(*******************************************************************************
                          protoc-gen-twincat V0.0.0.0                           
             https://github.bhs-world.com/CorrML/protoc-gen-twincat             
*******************************************************************************)
{attribute 'no_explicit_call' := 'do not call this POU directly'}
{attribute 'no-analysis'}
FUNCTION_BLOCK INTERNAL FINAL FB_ScalarTypes IMPLEMENTS I_Message
VAR
    _fbMessageParser : FB_MessageParser(ipMessage:= THIS^);
    _fbMessageWriter : FB_MessageWriter(ipMessage:= THIS^);
    _stScalarTypes : ST_ScalarTypes;
    END_VAR

{attribute 'no-analysis'}
(* Calculates the size of this message in Protocol Buffer wire format, in bytes. *)
METHOD CalculateSize : UDINT
VAR
    nSize : UDINT;
    nRepeatedFieldSize : UDINT;
END_VAR
// double double_value = 1;
nSize := nSize + 1 + F_ComputeDoubleSize(fValue:= _stScalarTypes.double_value);
// float float_value = 2;
nSize := nSize + 1 + F_ComputeFloatSize(fValue:= _stScalarTypes.float_value);
// int32 int32_value = 3;
nSize := nSize + 1 + F_ComputeInt32Size(anyDint:= _stScalarTypes.int32_value);
// int32 int32_value_as_word = 30;
nSize := nSize + 2 + F_ComputeInt32Size(anyDint:= _stScalarTypes.int32_value_as_word);
// int64 int64_value = 4;
nSize := nSize + 1 + F_ComputeInt64Size(anyLint:= _stScalarTypes.int64_value);
// int64 int64_value_as_dint = 40;
nSize := nSize + 2 + F_ComputeInt64Size(anyLint:= _stScalarTypes.int64_value_as_dint);
// uint32 uint32_value = 5;
nSize := nSize + 1 + F_ComputeUint32Size(anyUdint:= _stScalarTypes.uint32_value);
// uint32 uint32_value_as_byte = 50;
nSize := nSize + 2 + F_ComputeUint32Size(anyUdint:= _stScalarTypes.uint32_value_as_byte);
// uint64 uint64_value = 6;
nSize := nSize + 1 + F_ComputeUint64Size(anyUlint:= _stScalarTypes.uint64_value);
// uint64 uint64_value_as_dword = 60;
nSize := nSize + 2 + F_ComputeUint64Size(anyUlint:= _stScalarTypes.uint64_value_as_dword);
// sint32 sint32_value = 7;
nSize := nSize + 1 + F_ComputeSint32Size(anyDint:= _stScalarTypes.sint32_value);
// sint64 sint64_value = 8;
nSize := nSize + 1 + F_ComputeSint64Size(anyLint:= _stScalarTypes.sint64_value);
// fixed32 fixed32_value = 9;
nSize := nSize + 1 + F_ComputeFixed32Size(nValue:= _stScalarTypes.fixed32_value);
// fixed64 fixed64_value = 10;
nSize := nSize + 1 + F_ComputeFixed64Size(nValue:= _stScalarTypes.fixed64_value);
// sfixed32 sfixed32_value = 11;
nSize := nSize + 1 + F_ComputeSfixed32Size(nValue:= _stScalarTypes.sfixed32_value);
// sfixed64 sfixed64_value = 12;
nSize := nSize + 1 + F_ComputeSfixed64Size(nValue:= _stScalarTypes.sfixed64_value);
// bool bool_value = 13;
nSize := nSize + 1 + F_ComputeBoolSize(bValue:= _stScalarTypes.bool_value);
// string string_value = 14;
nSize := nSize + 1 + F_ComputeStringSize(anyString:= _stScalarTypes.string_value);
// bytes bytes_value = 15;
nSize := nSize + 1 + F_ComputeBytesSize(aBytes:= _stScalarTypes.bytes_value, nCount:= _stScalarTypes.bytes_value_count);
CalculateSize := nSize;
END_METHOD

(* Merges the data from the specified coded input stream with the current message.*)
METHOD MergeFrom : HRESULT
VAR_IN_OUT
    fbParseCtx : FB_ParseContext;
END_VAR
VAR
    nTag : UDINT;
END_VAR
REPEAT
MergeFrom := fbParseCtx.ReadTag(nTag=> nTag);
IF SUCCEEDED(MergeFrom) AND nTag = 0 THEN
    EXIT;
END_IF;

IF FAILED(MergeFrom) THEN
    RETURN;
END_IF

CASE nTag OF
    16#09:    // double double_value = 1;
        MergeFrom := fbParseCtx.ReadDouble(fValue=> _stScalarTypes.double_value); 
    16#15:    // float float_value = 2;
        MergeFrom := fbParseCtx.ReadFloat(fValue=> _stScalarTypes.float_value); 
    16#18:    // int32 int32_value = 3;
        MergeFrom := fbParseCtx.ReadInt32(anyDint:= _stScalarTypes.int32_value); 
    16#F0:    // int32 int32_value_as_word = 30;
        MergeFrom := fbParseCtx.ReadInt32(anyDint:= _stScalarTypes.int32_value_as_word); 
    16#20:    // int64 int64_value = 4;
        MergeFrom := fbParseCtx.ReadInt64(anyLint:= _stScalarTypes.int64_value); 
    16#140:    // int64 int64_value_as_dint = 40;
        MergeFrom := fbParseCtx.ReadInt64(anyLint:= _stScalarTypes.int64_value_as_dint); 
    16#28:    // uint32 uint32_value = 5;
        MergeFrom := fbParseCtx.ReadUint32(anyUdint:= _stScalarTypes.uint32_value); 
    16#190:    // uint32 uint32_value_as_byte = 50;
        MergeFrom := fbParseCtx.ReadUint32(anyUdint:= _stScalarTypes.uint32_value_as_byte); 
    16#30:    // uint64 uint64_value = 6;
        MergeFrom := fbParseCtx.ReadUint64(anyUlint:= _stScalarTypes.uint64_value); 
    16#1E0:    // uint64 uint64_value_as_dword = 60;
        MergeFrom := fbParseCtx.ReadUint64(anyUlint:= _stScalarTypes.uint64_value_as_dword); 
    16#38:    // sint32 sint32_value = 7;
        MergeFrom := fbParseCtx.ReadSint32(anyDint:= _stScalarTypes.sint32_value); 
    16#40:    // sint64 sint64_value = 8;
        MergeFrom := fbParseCtx.ReadSint64(anyLint:= _stScalarTypes.sint64_value); 
    16#4D:    // fixed32 fixed32_value = 9;
        MergeFrom := fbParseCtx.ReadFixed32(nValue=> _stScalarTypes.fixed32_value); 
    16#51:    // fixed64 fixed64_value = 10;
        MergeFrom := fbParseCtx.ReadFixed64(nValue=> _stScalarTypes.fixed64_value); 
    16#5D:    // sfixed32 sfixed32_value = 11;
        MergeFrom := fbParseCtx.ReadSfixed32(nValue=> _stScalarTypes.sfixed32_value); 
    16#61:    // sfixed64 sfixed64_value = 12;
        MergeFrom := fbParseCtx.ReadSfixed64(nValue=> _stScalarTypes.sfixed64_value); 
    16#68:    // bool bool_value = 13;
        MergeFrom := fbParseCtx.ReadBool(bValue=> _stScalarTypes.bool_value); 
    16#72:    // string string_value = 14;
        MergeFrom := fbParseCtx.ReadString(anyStringOut:= _stScalarTypes.string_value); 
    16#7A:    // bytes bytes_value = 15;
        MergeFrom := fbParseCtx.ReadBytes(aBytes:= _stScalarTypes.bytes_value, nCount=> _stScalarTypes.bytes_value_count); 
ELSE
    MergeFrom := fbParseCtx.SkipLastField();
END_CASE

UNTIL (FAILED(MergeFrom) OR nTag = 0)
END_REPEAT
END_METHOD

PROPERTY PUBLIC MessageValue : T_Any
GET
MessageValue := F_ToAnyType(anyArg:= _stScalarTypes);
END_GET
END_PROPERTY

PROPERTY PUBLIC Parser : REFERENCE TO FB_MessageParser
GET
Parser REF= THIS^._fbMessageParser;
END_GET
END_PROPERTY

PROPERTY PUBLIC ScalarTypes : ST_ScalarTypes
GET
ScalarTypes := _stScalarTypes;
END_GET
SET
_stScalarTypes := ScalarTypes;
END_SET
END_PROPERTY

(* Writer for this message.*)
PROPERTY PUBLIC Writer : REFERENCE TO FB_MessageWriter
GET
Writer REF= THIS^._fbMessageWriter;
END_GET
END_PROPERTY

(* Writes the data to the given coded output stream.*)
METHOD WriteTo : HRESULT
VAR_IN_OUT
	(* Coded output stream to write the data to. *)
	fbWriteCtx	: FB_WriteContext;
END_VAR
// double double_value = 1;
WriteTo := fbWriteCtx.WriteTag(1, E_WireType.Fixed64);
IF FAILED(WriteTo) THEN
    RETURN;
END_IF
WriteTo := fbWriteCtx.WriteDouble(fValue:= _stScalarTypes.double_value);
IF FAILED(WriteTo) THEN
    RETURN;
END_IF
// float float_value = 2;
WriteTo := fbWriteCtx.WriteTag(2, E_WireType.Fixed32);
IF FAILED(WriteTo) THEN
    RETURN;
END_IF
WriteTo := fbWriteCtx.WriteFloat(fValue:= _stScalarTypes.float_value);
IF FAILED(WriteTo) THEN
    RETURN;
END_IF
// int32 int32_value = 3;
WriteTo := fbWriteCtx.WriteTag(3, E_WireType.Varint);
IF FAILED(WriteTo) THEN
    RETURN;
END_IF
WriteTo := fbWriteCtx.WriteInt32(anyDint:= _stScalarTypes.int32_value);
IF FAILED(WriteTo) THEN
    RETURN;
END_IF
// int32 int32_value_as_word = 30;
WriteTo := fbWriteCtx.WriteTag(30, E_WireType.Varint);
IF FAILED(WriteTo) THEN
    RETURN;
END_IF
WriteTo := fbWriteCtx.WriteInt32(anyDint:= _stScalarTypes.int32_value_as_word);
IF FAILED(WriteTo) THEN
    RETURN;
END_IF
// int64 int64_value = 4;
WriteTo := fbWriteCtx.WriteTag(4, E_WireType.Varint);
IF FAILED(WriteTo) THEN
    RETURN;
END_IF
WriteTo := fbWriteCtx.WriteInt64(anyLint:= _stScalarTypes.int64_value);
IF FAILED(WriteTo) THEN
    RETURN;
END_IF
// int64 int64_value_as_dint = 40;
WriteTo := fbWriteCtx.WriteTag(40, E_WireType.Varint);
IF FAILED(WriteTo) THEN
    RETURN;
END_IF
WriteTo := fbWriteCtx.WriteInt64(anyLint:= _stScalarTypes.int64_value_as_dint);
IF FAILED(WriteTo) THEN
    RETURN;
END_IF
// uint32 uint32_value = 5;
WriteTo := fbWriteCtx.WriteTag(5, E_WireType.Varint);
IF FAILED(WriteTo) THEN
    RETURN;
END_IF
WriteTo := fbWriteCtx.WriteUint32(anyUdint:= _stScalarTypes.uint32_value);
IF FAILED(WriteTo) THEN
    RETURN;
END_IF
// uint32 uint32_value_as_byte = 50;
WriteTo := fbWriteCtx.WriteTag(50, E_WireType.Varint);
IF FAILED(WriteTo) THEN
    RETURN;
END_IF
WriteTo := fbWriteCtx.WriteUint32(anyUdint:= _stScalarTypes.uint32_value_as_byte);
IF FAILED(WriteTo) THEN
    RETURN;
END_IF
// uint64 uint64_value = 6;
WriteTo := fbWriteCtx.WriteTag(6, E_WireType.Varint);
IF FAILED(WriteTo) THEN
    RETURN;
END_IF
WriteTo := fbWriteCtx.WriteUint64(anyUlint:= _stScalarTypes.uint64_value);
IF FAILED(WriteTo) THEN
    RETURN;
END_IF
// uint64 uint64_value_as_dword = 60;
WriteTo := fbWriteCtx.WriteTag(60, E_WireType.Varint);
IF FAILED(WriteTo) THEN
    RETURN;
END_IF
WriteTo := fbWriteCtx.WriteUint64(anyUlint:= _stScalarTypes.uint64_value_as_dword);
IF FAILED(WriteTo) THEN
    RETURN;
END_IF
// sint32 sint32_value = 7;
WriteTo := fbWriteCtx.WriteTag(7, E_WireType.Varint);
IF FAILED(WriteTo) THEN
    RETURN;
END_IF
WriteTo := fbWriteCtx.WriteSint32(anyDint:= _stScalarTypes.sint32_value);
IF FAILED(WriteTo) THEN
    RETURN;
END_IF
// sint64 sint64_value = 8;
WriteTo := fbWriteCtx.WriteTag(8, E_WireType.Varint);
IF FAILED(WriteTo) THEN
    RETURN;
END_IF
WriteTo := fbWriteCtx.WriteSint64(anyLint:= _stScalarTypes.sint64_value);
IF FAILED(WriteTo) THEN
    RETURN;
END_IF
// fixed32 fixed32_value = 9;
WriteTo := fbWriteCtx.WriteTag(9, E_WireType.Fixed32);
IF FAILED(WriteTo) THEN
    RETURN;
END_IF
WriteTo := fbWriteCtx.WriteFixed32(nValue:= _stScalarTypes.fixed32_value);
IF FAILED(WriteTo) THEN
    RETURN;
END_IF
// fixed64 fixed64_value = 10;
WriteTo := fbWriteCtx.WriteTag(10, E_WireType.Fixed64);
IF FAILED(WriteTo) THEN
    RETURN;
END_IF
WriteTo := fbWriteCtx.WriteFixed64(nValue:= _stScalarTypes.fixed64_value);
IF FAILED(WriteTo) THEN
    RETURN;
END_IF
// sfixed32 sfixed32_value = 11;
WriteTo := fbWriteCtx.WriteTag(11, E_WireType.Fixed32);
IF FAILED(WriteTo) THEN
    RETURN;
END_IF
WriteTo := fbWriteCtx.WriteSfixed32(nValue:= _stScalarTypes.sfixed32_value);
IF FAILED(WriteTo) THEN
    RETURN;
END_IF
// sfixed64 sfixed64_value = 12;
WriteTo := fbWriteCtx.WriteTag(12, E_WireType.Fixed64);
IF FAILED(WriteTo) THEN
    RETURN;
END_IF
WriteTo := fbWriteCtx.WriteSfixed64(nValue:= _stScalarTypes.sfixed64_value);
IF FAILED(WriteTo) THEN
    RETURN;
END_IF
// bool bool_value = 13;
WriteTo := fbWriteCtx.WriteTag(13, E_WireType.Varint);
IF FAILED(WriteTo) THEN
    RETURN;
END_IF
WriteTo := fbWriteCtx.WriteBool(bValue:= _stScalarTypes.bool_value);
IF FAILED(WriteTo) THEN
    RETURN;
END_IF
// string string_value = 14;
WriteTo := fbWriteCtx.WriteTag(14, E_WireType.LengthDelimited);
IF FAILED(WriteTo) THEN
    RETURN;
END_IF
WriteTo := fbWriteCtx.WriteString(sStringToWrite:= _stScalarTypes.string_value);
IF FAILED(WriteTo) THEN
    RETURN;
END_IF
// bytes bytes_value = 15;
WriteTo := fbWriteCtx.WriteTag(15, E_WireType.LengthDelimited);
IF FAILED(WriteTo) THEN
    RETURN;
END_IF
WriteTo := fbWriteCtx.WriteBytes(aBytes:= _stScalarTypes.bytes_value, nCount:= _stScalarTypes.bytes_value_count);
IF FAILED(WriteTo) THEN
    RETURN;
END_IF
END_METHOD

END_FUNCTION_BLOCK

(* stored: Version 1.1.0.1
   POU FB_ScalarTypes: Id {c8090daf-a3df-4d62-beed-66b1b7ba6f95}, SpecialFunc None
   Method CalculateSize: Id {d5ada9c4-7ef6-4b93-84fd-c5f2e7c38b4d}
   Method MergeFrom: Id {2b762a1c-de4a-43d1-88ad-ee3a1833ce96}
   Property MessageValue: Id {0b51ec73-815d-46bc-94b2-7d504ea32214}
   Get Get: Id {63752e05-8193-4057-a1b7-5b68a4459ec1}
   Property Parser: Id {22fdabf9-616e-4780-93a9-e6955ee11359}
   Get Get: Id {654f3777-9faa-45f7-9002-cc1307c341ce}
   Property ScalarTypes: Id {ce4f1a4c-24d4-4d03-9d3e-176d0b6c9d5d}
   Get Get: Id {8b29ce64-e21c-4d83-a258-b5b95e904983}
   Set Set: Id {2daad220-9535-4004-a96d-277ccc64f28c}
   Property Writer: Id {ffa6ac61-94fe-4c33-9958-847d4e58ee49}
   Get Get: Id {33797eee-040f-4839-87a8-0d83ac3cda88}
   Method WriteTo: Id {88d35f46-975a-4636-b7cd-6b0441524ecb} *)
